PROGRAM pouMsgS1
VAR
	
	
	
END_VAR

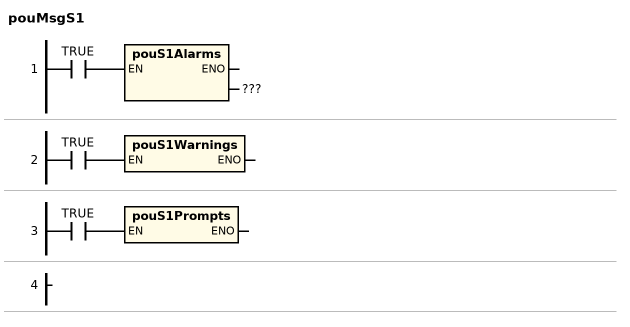
// NETWORK 1
pouS1Alarms();

// NETWORK 2
pouS1Warnings();

// NETWORK 3
pouS1Prompts();

// NETWORK 4

END_PROGRAM

(* stored: Version 1.1.0.1, ProductVersion 3.1.4024.12
   POU pouMsgS1: Id {71043ed9-688e-4f83-bc07-eae8159a6d6f}, SpecialFunc None *)
